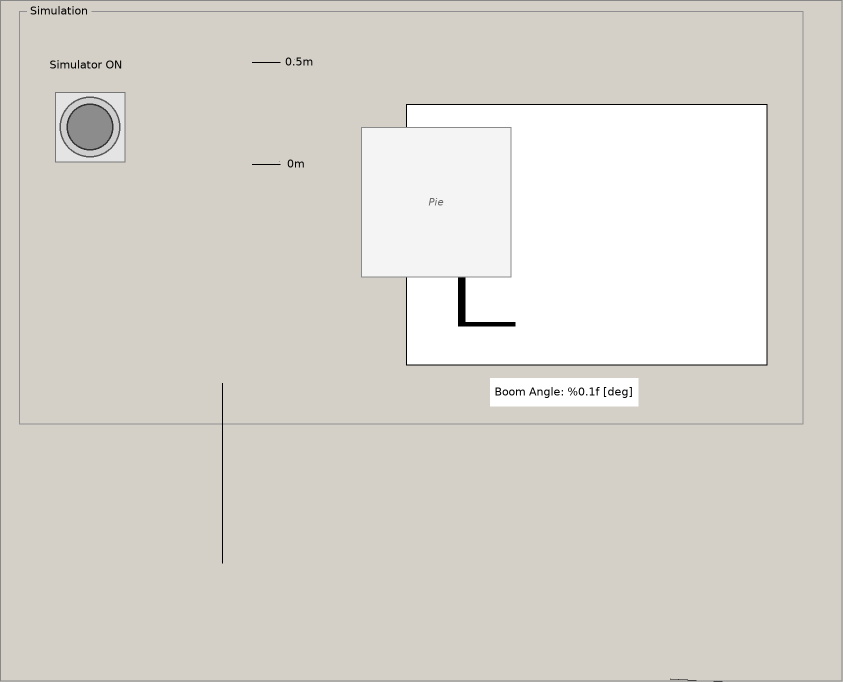
VISUALIZATION Animation  // 843x682
    GroupBox (19,3 784x421), "Simulation"
        Rectangle (387,101 361x261)
        Line (233,161) (261,161)
        Label (263,146 28x30), "0m"
        Line (233,59) (261,59)
        Textfield (470,374 150x30), "Boom Angle: %0.1f [deg]", text variable: G_Simulator.fBoomAngleDeg
        Rectangle (439,265 7x58)
        Rectangle (440,319 56x4)
        PushSwitch (36,89 70x70), variable: G_Simulator.bSimulatorOn, behaviour: TOGGLE, style: Switch-PushSwitch-Gray
    Line (222,383) (222,563)
        p1126004900: G_Simulator.stPistonAnimation.pt1_y
        p3528305787: G_Simulator.stPistonAnimation.pt0_x
        p2773130477: G_Simulator.stPistonAnimation.pt0_y
        p874137650: G_Simulator.stPistonAnimation.pt1_x
    Line (279,161) (279,161)
    Label (285,47 28x30), "0.5m"
    Line (294,59) (294,59)
    Line (722,682) (670,679)
        p1126004900: G_Simulator.stBoomAnimation.pt1_y
        p3528305787: G_Simulator.stBoomAnimation.pt0_x
        p2773130477: G_Simulator.stBoomAnimation.pt0_y
        p874137650: -G_Simulator.stBoomAnimation.pt1_x
    Label (-40,50 252x30), "Simulator ON"
    Pie (361,127 150x150)
END_VISUALIZATION

(* stored: Version 1.1.0.1, ProductVersion 3.1.4024.12
   Visu Animation: Id {4bdd8ed7-7379-4dd1-955f-a8a1c50d5ff4} *)
